{attribute 'OPC.UA.DA' := '1'}
{attribute 'OPC.UA.DA.StructuredType' := '1'}
TYPE BeamDiameterMsg :
STRUCT
	Id : EPowerIlluminationFlow;
	BeamDiameter : INT;
END_STRUCT
END_TYPE

(* stored: Version 1.1.0.1, ProductVersion 3.1.4024.3
   DUT BeamDiameterMsg: Id {3e400fac-26cf-40da-b0d9-fc607de12f50} *)
